SUBAPPLICATION Uebung_103 (* DigitalInput_I1 auf DigitalOutput_Q1, mit Plug and Socket *)
  (* Standard: 61499-2; Description: Copyright (c) 2023 Meisterschulen am Ostbahnhof This program and the accompanying materials are made available under the terms of the Eclipse Public License 2.0 which is available at https://www.eclipse.org/legal/epl-2.0/ SPDX-License-Identifier: EPL-2.0 *)
  (* Version 1.0, 2023-10-23, Franz Höpfinger, Meisterschulen am Ostbahnhof *)
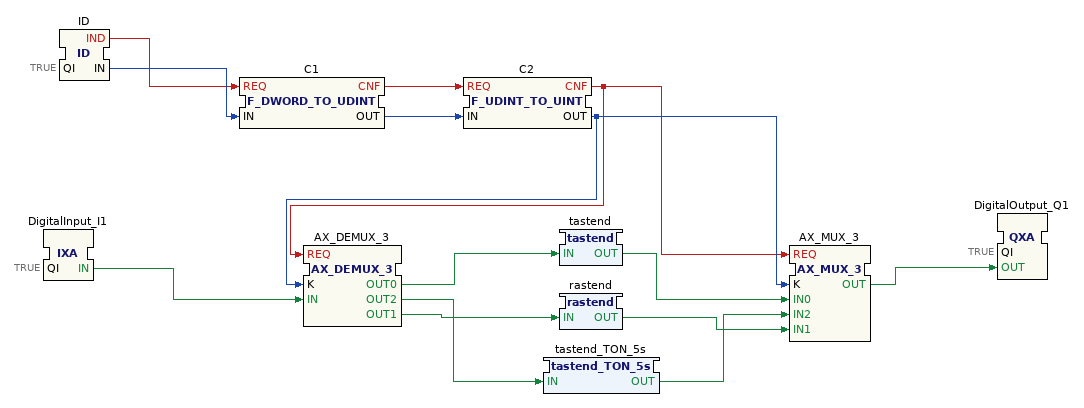
  FBS
    DigitalInput_I1 : IXA(QI := TRUE);
    DigitalOutput_Q1 : QXA(QI := TRUE);
    AX_DEMUX_3 : AX_DEMUX_3;
    AX_MUX_3 : AX_MUX_3;
    ID : ID(QI := TRUE);
    C1 : F_DWORD_TO_UDINT;
    C2 : F_UDINT_TO_UINT;
  END_FBS
  SUBAPPS
    rastend : FBs::Uebungen::Uebung_103::subapp::rastend;
    tastend : FBs::Uebungen::Uebung_103::subapp::tastend;
    tastend_TON_5s : FBs::Uebungen::Uebung_103::subapp::tastend_TON_5s;
  END_SUBAPPS
  EVENT_CONNECTIONS
    ID.IND TO C1.REQ;
    C1.CNF TO C2.REQ;
    C2.CNF TO AX_DEMUX_3.REQ;
    C2.CNF TO AX_MUX_3.REQ;
  END_CONNECTIONS
  DATA_CONNECTIONS
    ID.IN TO C1.IN;
    C1.OUT TO C2.IN;
    C2.OUT TO AX_DEMUX_3.K;
    C2.OUT TO AX_MUX_3.K;
  END_CONNECTIONS
  ADAPTER_CONNECTIONS
    AX_MUX_3.OUT TO DigitalOutput_Q1.OUT;
    DigitalInput_I1.IN TO AX_DEMUX_3.IN;
    AX_DEMUX_3.OUT0 TO tastend.IN;
    tastend.OUT TO AX_MUX_3.IN0;
    AX_DEMUX_3.OUT2 TO tastend_TON_5s.IN;
    tastend_TON_5s.OUT TO AX_MUX_3.IN2;
    rastend.OUT TO AX_MUX_3.IN1;
    AX_DEMUX_3.OUT1 TO rastend.IN;
  END_CONNECTIONS
END_SUBAPPLICATION
